(*

## Short summary
An implementation of the ``ISinlgeExecutionCycleManager`` to provide simple cycle managment for steps in state machines.
The body NEEDS to be called at the start of every cycle (before using the step property) ONLY ONCE.

.. <info>
If used in the same step, the order of method calls should be this:
configurations
enter
executeCommand
evaluate
waitFor
proceed
proceedWith
acknowledge
leave
.. </info>

.. <legal notes>

legal notes
=================
| SPDX-FileCopyrightText: © 2024 ekvip automation GmbH <info@ekvip.de>
| SPDX-License-Identifier: Apache-2.0
| For details check: Apache-2.0_

.. _Apache-2.0: https://www.apache.org/licenses/LICENSE-2.0

.. </legal notes>



*)
FUNCTION_BLOCK SimpleCycleManager EXTENDS AbstractCycleManager
VAR_INPUT
	(*control bit to start or abort the cycle manager*)
	execute :BOOL;
	(*used for StopRequest evaluation if configured*)
	stopRequest :BOOL := FALSE;
	(*if true and Pausing Enabled and busy will proceed with PAUSE*)
	pause :BOOL := FALSE;
	(*if true, will acknowledge error and return to previous step*)
	resume :BOOL := FALSE;
	(* must be TRUE if stepping is enabled to proceed steps automatically *)
	stepControl :BOOL := TRUE;
END_VAR

THIS^.update(
	execute := execute, 
	pause := pause, 
	resume := resume, 
	stepControl := stepControl, 
	stopRequest := stopRequest
);

(*

## Short summary
This abstract property returns the class name of the concrete object, 
which is useful for logging/debugging purpose or to check the class name
for ``__DELETE`` in factories (sometimes it's necessary to do more 
than just to free the memory).

.. <legal notes>

legal notes
=================
| SPDX-FileCopyrightText: © 2022 ekvip automation GmbH <info@ekvip.de>
| SPDX-License-Identifier: Apache-2.0
| For details check: Apache-2.0_

.. _Apache-2.0: https://www.apache.org/licenses/LICENSE-2.0

.. </legal notes>

*)
PROPERTY className : CNM_AbstractObject.ClassName
GET
className := 'CNM_CycleManager.SimpleCycleManager';
END_GET
END_PROPERTY

END_FUNCTION_BLOCK

(* stored: Version 1.1.0.1
   POU SimpleCycleManager: Id {7625fde4-248d-4e82-a884-39cfee5f0a69}, SpecialFunc None
   Property className: Id {fa19b843-eb5b-4493-bbe8-50b1a509fd78}
   Get Get: Id {5fa77345-bcf8-4ec1-9c15-ed1b0f7957ed} *)
